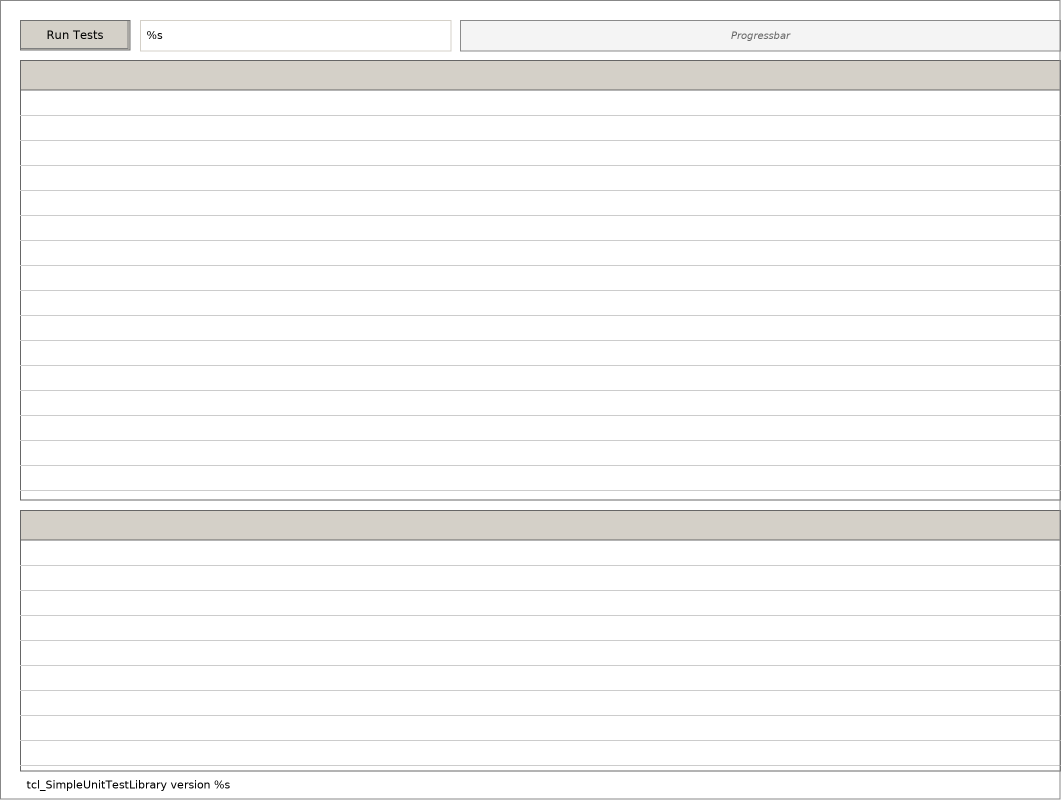
VISUALIZATION Visualization  // 1061x800
    Button (20,20 110x30), "Run Tests"
        tap TestFramework.TestRunner.Run
    Textfield (140,20 311x31), "%s", text variable: TestFramework.TestRunner._Results
    Table (20,60 1041x440), data array: TestFramework.TestRunner.TestResults
        p2170511999: TestFramework.TestRunner.TestResults[INDEX].ImageRef
        p1755163831: Test State
        p338671338: TestFramework.TestRunner.TestResults[INDEX].TestState
        p511219082: Test Name
        p1892666644: TestFramework.TestRunner.TestResults[INDEX].TestName
        p2232123230: Time
        p3854506369: TestFramework.TestRunner.TestResults[INDEX].TestCompleteTime
    Table (20,510 1041x261), data array: TestFramework.TestRunner.AssertionMessages._Messages
        p3854506369: TestFramework.TestRunner.AssertionMessages._Messages[INDEX]
        p2232123230: Assertion Messages
    Progressbar (460,20 601x31), variable: TestFramework.TestRunner.TestsCompletedPercentage
    Rectangle (20,770 650x30), "tcl_SimpleUnitTestLibrary version %s", text variable: Global_Version.stLibVersion_tcl_SimpleUnitTestLibrary.sVersion
END_VISUALIZATION

(* stored: Version 1.1.0.1, ProductVersion 3.1.4024.4
   Visu Visualization: Id {deef92dd-c8d0-4c0a-b471-21d2af44be99} *)
